// TIA Portal V18 export
DATA_BLOCK "AutoProcessData_Buffer_Clear"   // DB1602
{ S7_Optimized_Access := 'FALSE' }
// stored: AutoNumber false
   VAR RETAIN
      DataBuffer : Array[0..60] of "ProcessDatad";
      DataBufferClear : "ProcessDatad";
      VAL { S7_SetPoint := 'True'} : Int;
   END_VAR
BEGIN
END_DATA_BLOCK
